FUNCTION_BLOCK EL2044
VAR
	{attribute addProperty Name "WcState"}
	_wcState : WcStateInputToggle;
	{attribute addProperty Name "Info data"}
	_infoData : InfoDataAds;
	_io : EL2044_Data;
END_VAR

PROPERTY IO : REFERENCE TO EL2044_Data
GET
IO REF= _io;
END_GET
END_PROPERTY

PROPERTY WcState : REFERENCE TO WcStateInputToggle
GET
WcState REF= _wcState;
END_GET
END_PROPERTY

END_FUNCTION_BLOCK

(* stored: Version 1.1.0.1, ProductVersion 3.1.4024.9
   POU EL2044: Id {294e1e75-1edd-0b24-34ca-30044f55b5db}, SpecialFunc None
   Property IO: Id {041d236d-cc09-02f0-18d0-84f96a2561ac}
   Get Get: Id {30daf7e6-d456-0bd1-35ef-6d13d00ada7e}
   Property WcState: Id {ee72c114-a2c3-04ee-3c44-19031c86d5d3}
   Get Get: Id {e26fc1ca-f550-06ec-1477-3cd6df0b8135} *)
